SUBAPPLICATION Uebung_012a_sub (* Numeric Value Input und Speichern *)
  (* Standard: 61499-2; Description: Copyright (c) 2023 Meisterschulen am Ostbahnhof This program and the accompanying materials are made available under the terms of the Eclipse Public License 2.0 which is available at https://www.eclipse.org/legal/epl-2.0/ SPDX-License-Identifier: EPL-2.0 *)
  (* Version 1.0, 2023-10-31, Franz Höpfinger, Meisterschulen am Ostbahnhof *)
  IMPORT logiBUS::io::DI::logiBUS_DI;
  IMPORT logiBUS::io::DI::logiBUS_DI_Events;
  IMPORT logiBUS::io::DQ::logiBUS_DO;
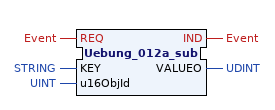
  EVENT_INPUT
    REQ;
  END_EVENT
  EVENT_OUTPUT
    IND;
  END_EVENT
  VAR_INPUT
    KEY : STRING;
    u16ObjId : UINT;
  END_VAR
  VAR_OUTPUT
    VALUEO : UDINT;
  END_VAR
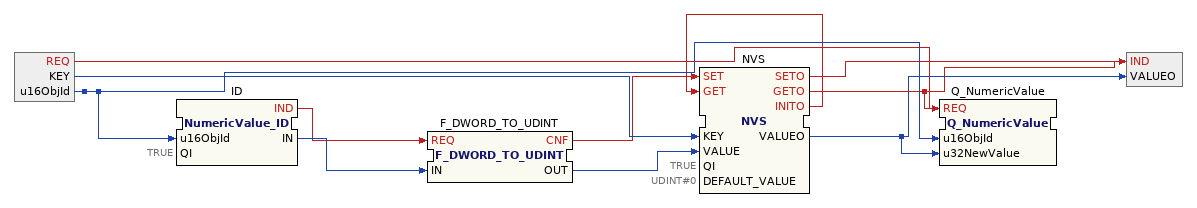
  FBS
    ID : NumericValue_ID(QI := TRUE);
    F_DWORD_TO_UDINT : F_DWORD_TO_UDINT;
    NVS : NVS(QI := TRUE, DEFAULT_VALUE := UDINT#0);
    Q_NumericValue : isobus::ut::Q_NumericValue;
  END_FBS
  EVENT_CONNECTIONS
    ID.IND TO F_DWORD_TO_UDINT.REQ;
    REQ TO Q_NumericValue.REQ;
    F_DWORD_TO_UDINT.CNF TO NVS.SET;
    NVS.SETO TO IND;
    NVS.GETO TO Q_NumericValue.REQ;
    NVS.GETO TO IND;
    NVS.INITO TO NVS.GET;
  END_CONNECTIONS
  DATA_CONNECTIONS
    ID.IN TO F_DWORD_TO_UDINT.IN;
    u16ObjId TO Q_NumericValue.u16ObjId;
    KEY TO NVS.KEY;
    F_DWORD_TO_UDINT.OUT TO NVS.VALUE;
    NVS.VALUEO TO Q_NumericValue.u32NewValue;
    NVS.VALUEO TO VALUEO;
    u16ObjId TO ID.u16ObjId;
  END_CONNECTIONS
END_SUBAPPLICATION
